FUNCTION_BLOCK FB_SortingSystem_TSM EXTENDS FB_TSM
VAR
	fbConveyorEM			: FB_Conveyor_EM;

	ButtonFaultReset    AT %I* : BOOL;
    ButtonStartProceed  AT %I* : BOOL;
    ButtonAbort         AT %I* : BOOL;
	ButtonRun			AT %I* : BOOL;
END_VAR

SUPER^();

// System Interlocks
    // The system interlock inherits the system interlock from the TSM's EMs OR from the safety zone. More interlocks can be added that are not part of the EM or safety zone interlocks.  
    SUPER^.P_SystemInterlock.M_Set(Index := 0, Description := 'Always TRUE' , Condition := TRUE);   // network devices OK

// Button Requests
    IF ButtonFaultReset THEN
        ButtonFaultReset := FALSE;
        SUPER^.M_Retry();
    ELSIF ButtonStartProceed THEN
        ButtonStartProceed := FALSE;
        SUPER^.M_Proceed();
    ELSIF ButtonAbort THEN
        ButtonAbort := FALSE;
        SUPER^.M_Abort();
    END_IF

// State Permissives
// Start
    SUPER^.P_StartPermissive.M_Set(index := 0, Description := 'FlipGantryEM in Fixed State', Condition := fbConveyorEM.P_Status.FixedStateIndex <> 0);
// Home
    SUPER^.P_HomePermissive.M_Set(index := 0, Description := 'Always TRUE', Condition := TRUE);
// Proceed
    SUPER^.P_ProceedPermissive.M_Set(index := 0, Description := 'Always TRUE', Condition := TRUE);

// Retry EMs on TSM Retry
    IF SUPER^.P_Status.Retry THEN
        fbConveyorEM.M_Retry();
	END_IF

// Equipment Modules
	M_ConveyorEM();

METHOD PROTECTED _M_Aborting
// Abort child Equipment Modules
    fbConveyorEM.M_Abort();

// Aborting Complete Permissives - Method will be cyclically executed until all permissives are met
    SUPER^.P_AbortCompletePermissive.M_Set(Index := 0,
										   Description := 'Conveyor Aborted',
										   Condition := fbConveyorEM.P_Status.StateStatus <> E_DeviceStatus.Active OR
														fbConveyorEM.P_Status.StateStatus <> E_DeviceStatus.Aborting);
END_METHOD

METHOD PROTECTED _M_Homing
//=========================================================================================
//    local constants
//=========================================================================================
VAR CONSTANT
    START                                                       : UDINT := 10;       // 10

    COMPLETE                                                    : UDINT := 1000;     // 1000
END_VAR
//=========================================================================================
//    local variables
//=========================================================================================
VAR_INST
    
END_VAR
// Set first step to 10
SUPER^.P_Configuration.HomingFirstStep := 10;

CASE SUPER^.P_HomingSequencer.P_Status.CurrentStep OF
	START:
        // Branch 0: At fixed state, skip PalletPositioner recovery and Finish
		SUPER^.P_HomingSequencer.M_SetBranchConfig(BranchIndex := 0, Description := 'No Recovery Needed', NextStep := COMPLETE, CheckWhileFaulted := TRUE);
		SUPER^.P_HomingSequencer.M_SetBranchPermissive(BranchIndex := 0,
                                                        PermissiveIndex := 0,
                                                        Description := 'At Fixed State',
                                                        Condition := fbConveyorEM.P_Status.FixedStateIndex <> 0);
	COMPLETE:
		_M_SeqComplete();
END_CASE
END_METHOD

METHOD PROTECTED _M_Pausing
VAR CONSTANT
    COMMAND_PAUSE : UDINT := 10;
	FINISH        : UDINT := 999;
END_VAR
// Set first step to 10
SUPER^.P_Configuration.PausingFirstStep := 10;

// Pausing Sequence
CASE SUPER^.P_PausingSequencer.P_Status.CurrentStep OF	
	COMMAND_PAUSE:
		CASE SUPER^.P_PausingSequencer.P_StepStatus.StepState OF
			E_StepState.ActiveEntry:
                // Set step configurations here
                SUPER^.P_PausingSequencer.P_StepConfig.Name := 'Pause EMs';
				SUPER^.P_PausingSequencer.P_StepConfig.Timeout := T#15S; // Optional step timeout. Set to zero to ignore
                // Issue EM commands here
				    fbConveyorEM.M_Pause();
			E_StepState.ActiveDuring:
                // Check for errors on EMs commanded on this step here
				SUPER^.P_PausingSequencer.M_CheckFaultCondition(Error := fbConveyorEM.P_Error);
            E_StepState.ActiveExit:
                //
            E_StepState.FaultedEntry:
                //
            E_StepState.FaultedDuring:
                //
            E_StepState.FaultedExit:
                //
        END_CASE
        // Branch 0: EMs Paused Successfully
		SUPER^.P_PausingSequencer.M_SetBranchConfig(BranchIndex := 0, Description := 'EMs Paused Successfully', NextStep := FINISH, CheckWhileFaulted := TRUE);
		SUPER^.P_PausingSequencer.M_SetBranchPermissive(BranchIndex := 0,
                                                           PermissiveIndex := 0,
                                                           Description := 'fbConveyorEM Paused OR Complete',
                                                           Condition := fbConveyorEM.P_Status.StateStatus = E_DeviceStatus.Paused OR
                                                                        fbConveyorEM.P_Status.StateStatus = E_DeviceStatus.Complete);                                                 
        
	FINISH:
        // Sequence must end with the following method call
		_M_SeqComplete(); 
END_CASE
END_METHOD

METHOD PROTECTED _M_Proceeding
VAR CONSTANT
    COMMAND_PROCEED : UDINT := 10;
	FINISH          : UDINT := 999;
END_VAR
// Set first step to 10
SUPER^.P_Configuration.ProceedingFirstStep := 10;

// Proceeding Sequence
CASE SUPER^.P_ProceedingSequencer.P_Status.CurrentStep OF	
	COMMAND_PROCEED:
		CASE SUPER^.P_ProceedingSequencer.P_StepStatus.StepState OF
			E_StepState.ActiveEntry:
                // Set step configurations here
                SUPER^.P_ProceedingSequencer.P_StepConfig.Name := 'Proceed EMs';
				SUPER^.P_ProceedingSequencer.P_StepConfig.Timeout := T#15S; // Optional step timeout. Set to zero to ignore
                // Issue EM commands here
				    fbConveyorEM.M_Proceed();
			E_StepState.ActiveDuring:
                // Check for errors on EMs commanded on this step here
				SUPER^.P_ProceedingSequencer.M_CheckFaultCondition(Error := fbConveyorEM.P_Error);
            E_StepState.ActiveExit:
                //
            E_StepState.FaultedEntry:
                //
            E_StepState.FaultedDuring:
                //
            E_StepState.FaultedExit:
                //
        END_CASE
        // Branch 0: EMs Proceeded Successfully
		SUPER^.P_ProceedingSequencer.M_SetBranchConfig(BranchIndex := 0, Description := 'EMs Proceeded Successfully', NextStep := FINISH, CheckWhileFaulted := TRUE);
		SUPER^.P_ProceedingSequencer.M_SetBranchPermissive(BranchIndex := 0,
                                                           PermissiveIndex := 0,
                                                           Description := 'fbConveyorEM Active OR Complete',
                                                           Condition := fbConveyorEM.P_Status.StateStatus = E_DeviceStatus.Active OR
                                                                        fbConveyorEM.P_Status.StateStatus = E_DeviceStatus.Complete);                                                    
        
	FINISH:
        // Sequence must end with the following method call
		_M_SeqComplete(); 
END_CASE
END_METHOD

METHOD PROTECTED _M_Running
VAR CONSTANT
    START_BRANCH	: UDINT := 10;
    START			: UDINT := 20;
	RUNNING			: UDINT := 30;
	STOP			: UDINT := 40;
	FINISH			: UDINT := 999;
END_VAR
// Set first step to 10
SUPER^.P_Configuration.RunningFirstStep := 10;

CASE SUPER^.P_RunningSequencer.P_Status.CurrentStep OF
	START_BRANCH:
        // Branch 0:
		SUPER^.P_RunningSequencer.M_SetBranchConfig(BranchIndex := 0, Description := 'Conveyor START', NextStep := START, CheckWhileFaulted := TRUE);
		SUPER^.P_RunningSequencer.M_SetBranchPermissive(BranchIndex := 0,
                                                        PermissiveIndex := 0,
                                                        Description := 'EM at Stopped',
                                                        Condition := fbConveyorEM.P_Status.FixedStateIndex = E_ConveyorEMFixed.Stopped);
		SUPER^.P_RunningSequencer.M_SetBranchPermissive(BranchIndex := 0,
                                                        PermissiveIndex := 1,
                                                        Description := 'ButtonRun is TRUE',
                                                        Condition := ButtonRun);

        // Branch 1:
		SUPER^.P_RunningSequencer.M_SetBranchConfig(BranchIndex := 1, Description := 'Conveyor Running', NextStep := RUNNING, CheckWhileFaulted := TRUE);
		SUPER^.P_RunningSequencer.M_SetBranchPermissive(BranchIndex := 1,
                                                        PermissiveIndex := 0,
                                                        Description := 'EM at Running',
                                                        Condition := fbConveyorEM.P_Status.FixedStateIndex = E_ConveyorEMFixed.Running);
    START:
        CASE SUPER^.P_RunningSequencer.P_StepStatus.StepState OF
			E_StepState.ActiveEntry:
                // Set step configurations here
                SUPER^.P_RunningSequencer.P_StepConfig.Name := 'Command EM to Run Conveyor';
				SUPER^.P_RunningSequencer.P_StepConfig.Timeout := T#5S; // Optional step timeout. Set to zero to ignore
                SUPER^.P_RunningSequencer.P_StepConfig.IgnoreHold := FALSE; // This step is pausable.
                SUPER^.P_RunningSequencer.P_StepConfig.NextStepAfterRetry := 0; // Optional.  Set to zero to ignore
                // Issue EM commands here
                    fbConveyorEM.M_TransitionNumberRequest(E_ConveyorEMTransition.Starting);
			E_StepState.ActiveDuring:
                // Check for errors on EMs commanded on this step here
                SUPER^.P_RunningSequencer.M_CheckFaultCondition(Error := fbConveyorEM.P_Error);
            E_StepState.ActiveExit:
                //
            E_StepState.FaultedEntry:
                //
            E_StepState.FaultedDuring:
                //
            E_StepState.FaultedExit:
                //
        END_CASE
		// Branch 0: EMs Proceeded Successfully
		SUPER^.P_RunningSequencer.M_SetBranchConfig(BranchIndex := 0, Description := 'ConveyorEM Transition Finished', NextStep := RUNNING, CheckWhileFaulted := TRUE);
		SUPER^.P_RunningSequencer.M_SetBranchPermissive(BranchIndex := 0,
                                                        PermissiveIndex := 0,
                                                        Description := 'EM at Running',
                                                        Condition := fbConveyorEM.P_Status.FixedStateIndex = E_ConveyorEMFixed.Running);
    RUNNING:
        CASE SUPER^.P_RunningSequencer.P_StepStatus.StepState OF
			E_StepState.ActiveEntry:
                // Set step configurations here
                SUPER^.P_RunningSequencer.P_StepConfig.Name := 'Command EM to Run Conveyor';
				SUPER^.P_RunningSequencer.P_StepConfig.Timeout := T#0S; // Optional step timeout. Set to zero to ignore
                SUPER^.P_RunningSequencer.P_StepConfig.IgnoreHold := FALSE; // This step is pausable.
                SUPER^.P_RunningSequencer.P_StepConfig.NextStepAfterRetry := 0; // Optional.  Set to zero to ignore
                // Issue EM commands here
			E_StepState.ActiveDuring:
                // Check for errors on EMs commanded on this step here
                SUPER^.P_RunningSequencer.M_CheckFaultCondition(Error := fbConveyorEM.P_Error);
            E_StepState.ActiveExit:
                //
            E_StepState.FaultedEntry:
                //
            E_StepState.FaultedDuring:
                //
            E_StepState.FaultedExit:
                //
        END_CASE
		// Branch 0: EMs Proceeded Successfully
		SUPER^.P_RunningSequencer.M_SetBranchConfig(BranchIndex := 0, Description := 'TSM Received Complete Signal', NextStep := STOP, CheckWhileFaulted := TRUE);
		SUPER^.P_RunningSequencer.M_SetBranchPermissive(BranchIndex := 0,
                                                        PermissiveIndex := 0,
                                                        Description := 'ButtonRun is FALSE',
                                                        Condition := NOT ButtonRun);
    STOP:
        CASE SUPER^.P_RunningSequencer.P_StepStatus.StepState OF
			E_StepState.ActiveEntry:
                // Set step configurations here
                SUPER^.P_RunningSequencer.P_StepConfig.Name := 'Command EM to Run Conveyor';
				SUPER^.P_RunningSequencer.P_StepConfig.Timeout := T#5S; // Optional step timeout. Set to zero to ignore
                SUPER^.P_RunningSequencer.P_StepConfig.IgnoreHold := FALSE; // This step is pausable.
                SUPER^.P_RunningSequencer.P_StepConfig.NextStepAfterRetry := 0; // Optional.  Set to zero to ignore
                // Issue EM commands here
                    fbConveyorEM.M_TransitionNumberRequest(E_ConveyorEMTransition.Stopping);
			E_StepState.ActiveDuring:
                // Check for errors on EMs commanded on this step here
                SUPER^.P_RunningSequencer.M_CheckFaultCondition(Error := fbConveyorEM.P_Error);
            E_StepState.ActiveExit:
                //
            E_StepState.FaultedEntry:
                //
            E_StepState.FaultedDuring:
                //
            E_StepState.FaultedExit:
                //
        END_CASE
		// Branch 0: EMs Proceeded Successfully
		SUPER^.P_RunningSequencer.M_SetBranchConfig(BranchIndex := 0, Description := 'ConveyorEM Transition Finished', NextStep := FINISH, CheckWhileFaulted := TRUE);
		SUPER^.P_RunningSequencer.M_SetBranchPermissive(BranchIndex := 0,
                                                        PermissiveIndex := 0,
                                                        Description := 'EM at Stopped',
                                                        Condition := fbConveyorEM.P_Status.FixedStateIndex = E_ConveyorEMFixed.Stopped);
	FINISH:
        // Sequence must end with the following method call
		_M_SeqComplete(); 
END_CASE
END_METHOD

METHOD M_ConveyorEM
// Set System Interlocks
// Index 0 is set in EM FB

// Call EM
    fbConveyorEM();
END_METHOD

END_FUNCTION_BLOCK

(* stored: Version 1.1.0.1, ProductVersion 3.1.4024.6
   POU FB_SortingSystem_TSM: Id {f9741123-7b69-44b4-8663-6344edae9ebe}, SpecialFunc None
   Folder Equipment Modules: Id {96c199b6-20e6-4705-814f-d7d19ae55b93}
   Method _M_Aborting: Id {8f9bdb77-f42a-4993-b418-89ebbdbe8984}
   Method _M_Homing: Id {e934b0ae-fe24-417b-9f36-1c429a5e40a6}
   Method _M_Pausing: Id {d378e491-b1bd-4e62-a8fb-e98adba2e8d2}
   Method _M_Proceeding: Id {f1eaf918-cb4e-4418-af2f-37ab00ae53f9}
   Method _M_Running: Id {ae1be1e2-42ee-4656-b3b8-7841ed3d9e9e}
   Method M_ConveyorEM: Id {fecb3ecc-8902-4fb7-833c-fbaa8f6903cd} *)
